(* IEC 61131-3 sources: conversion/src/times, 5 files *)

(* ---- types.st ---- *)
NAMESPACE Simatic.Ax.Conversion.Times

    TYPE
        SimotionDateTime : STRUCT
            SimotionDate : DWORD;
            SimotionTime : DWORD;
        END_STRUCT;
    END_TYPE

END_NAMESPACE

(* ---- LDateAndTimeToSimotionDateToD.st ---- *)
USING System.DateTime;
NAMESPACE Simatic.Ax.Conversion.Times
    FUNCTION LDateAndTimeToSimotionDateTime
        VAR_INPUT
            SimaticTime : LDATE_AND_TIME;
        END_VAR
        VAR_OUTPUT
            SimotionTime : DWORD;
            SimotionDate : DWORD;
        END_VAR

        VAR_TEMP
            actDays : INT;
            actMonth : INT;
            actYear : INT;
            actHour : INT;
            actMinute : INT;
            actSecond : INT;
            actMillisecond : INT;
            elapsedYears : INT;
            elapsedDays : DINT;
            loop : DINT;
        END_VAR

        //we ignore microseconds and nanoseconds, since they are supported by the destination data type
        SplitDateAndTime(value := SimaticTime,
        year => actYear,
        month => actMonth,
        day => actDays,
        hour => actHour,
        minute => actMinute,
        second => actSecond,
        millisecond => actMillisecond);

        //add number of days from full years, subtracting the current year
        FOR loop := 1992 TO (actYear - 1) DO
            IF loop MOD 4 = 0 AND loop <> 2100 THEN
                elapsedDays := elapsedDays + 366;
            ELSE
                elapsedDays := elapsedDays + 365;
            END_IF;
        END_FOR;

        //add days from full months of the current year
        IF actMonth > 1 THEN
            elapsedDays := elapsedDays + 31;
        END_IF;
        IF actMonth > 2 THEN
            IF actYear MOD 4 = 0 AND NOT (actYear = 2100) THEN
                elapsedDays := elapsedDays + 29;
            ELSE
                elapsedDays := elapsedDays + 28;
            END_IF;
        END_IF;
        IF actMonth > 3 THEN
            elapsedDays := elapsedDays + 31;
        END_IF;
        IF actMonth > 4 THEN
            elapsedDays := elapsedDays + 30;
        END_IF;
        IF actMonth > 5 THEN
            elapsedDays := elapsedDays + 31;
        END_IF;
        IF actMonth > 6 THEN
            elapsedDays := elapsedDays + 30;
        END_IF;
        IF actMonth > 7 THEN
            elapsedDays := elapsedDays + 31;
        END_IF;
        IF actMonth > 8 THEN
            elapsedDays := elapsedDays + 31;
        END_IF;
        IF actMonth > 9 THEN
            elapsedDays := elapsedDays + 30;
        END_IF;
        IF actMonth > 10 THEN
            elapsedDays := elapsedDays + 31;
        END_IF;
        IF actMonth > 11 THEN
            elapsedDays := elapsedDays + 30;
        END_IF;

        //add days from current month
        elapsedDays := elapsedDays + actDays;

        SimotionDate := TO_DWORD(elapsedDays);
        SimotionTime := TO_DWORD (TO_UDINT(actMillisecond) + UDINT#1000 * (TO_UDINT(actSecond) + UDINT#60 * (TO_UDINT(actMinute + 60 * ( actHour)))));

    END_FUNCTION

END_NAMESPACE

(* ---- SimotionDateToDToLDateAndTime.st ---- *)
USING System.DateTime;
NAMESPACE Simatic.Ax.Conversion.Times

    FUNCTION SimotionDateTimeToLDateAndTime : LDATE_AND_TIME

        VAR_INPUT
         SimotionTime : DWORD;
         SimotionDate : DWORD;
        END_VAR

        VAR_TEMP
           u32Date : UDINT;
           u32Year : UDInt;
           u32Month : UDInt;
           u32Days : UDInt;
           b32AuxHours : UDInt;
           boDateReady : Bool;
           HOUR : UDINT;
           MINUTE : UDINT;
           SECOND : UDINT;
           NANOSECOND : UDINT;
        END_VAR

        u32Date := TO_UDINT(SimotionDate);// + UDINT#1;

         // calculation of hours
         HOUR := TO_UDINT(SimotionTime) / UDINT#3600000;
         b32AuxHours := TO_UDINT(SimotionTime) - HOUR * UDINT#3600000;

         // calculation of minutes
         MINUTE := b32AuxHours / UDINT#60000;

         // calculation of seconds
         SECOND :=  (b32AuxHours - MINUTE * UDINT#60000) / UDINT#1000;

         // calculation of mseconds
         NANOSECOND := ( TO_UDINT(SimotionTime) - (HOUR *  UDINT#3600000) - (MINUTE *  UDINT#60000) - (SECOND *  UDINT#1000)) *  UDINT#1000000;

         //Reset values to calculate actual year
         u32Year :=  UDINT#1991;
         u32Days :=  UDINT#0;

         //Detect actual year by adding the days since 01.01.1992
         REPEAT
           //Increase number of years
           u32Year := u32Year +  UDINT#1;
           //If year is a leap-year
           IF  (u32Year MOD  UDINT#4 =  UDINT#0) AND  (u32Year <>  UDINT#2100) THEN //only 2100 is not a leap-year between 1992-2200
             u32Days := u32Days +  UDINT#366;
           ELSE
             u32Days := u32Days +  UDINT#365;
           END_IF;
           //Number of days is greater or equals number of days of SIMOTION system
         UNTIL u32Days >= u32Date
         END_REPEAT;

         u32Days := u32Days;

         //Decrease number of days by number of days of one year
         //If year is a leap-year
         IF  (u32Year MOD  UDINT#4 =  UDINT#0) AND  (u32Year <>  UDINT#2100) THEN //only 2100 is not a leap-year between 1992-2200
           u32Date := u32Date -  (u32Days -  UDINT#366);
         ELSE
           u32Date := u32Date -  (u32Days -  UDINT#365);
         END_IF;

         //Reset values to calculate actual month and day
         u32Month :=  UDINT#1;
         boDateReady := FALSE;

         //Start CASE with value "1" (-> january)
         REPEAT
           CASE u32Month OF
               // for months with 31 days
               UDINT#1,  UDINT#3,  UDINT#5,  UDINT#7,  UDINT#8,  UDINT#10:
               IF  (u32Date <=  UDINT#31) THEN
                 u32Days := u32Date;
                 boDateReady := TRUE;
               ELSE
                 u32Month := u32Month +  UDINT#1;
                 u32Date := u32Date -  UDINT#31;
               END_IF;
               //for february
               UDINT#2:
               IF  (u32Year MOD  UDINT#4 =  UDINT#0) AND  (u32Year <>  UDINT#2100) THEN //only 2100 is not a leap-year between 1992-2200
                 IF  (u32Date <=  UDINT#29) THEN
                   u32Days := u32Date;
                   boDateReady := TRUE;
                 ELSE
                   u32Month := u32Month +  UDINT#1;
                   u32Date := u32Date -  UDINT#29;
                 END_IF;
               ELSE
                 IF  (u32Date <=  UDINT#28) THEN
                   u32Days := u32Date;
                   boDateReady := TRUE;
                 ELSE
                   u32Month := u32Month +  UDINT#1;
                   u32Date := u32Date -  UDINT#28;
                 END_IF;
               END_IF;
               //for months with 30 days
               UDINT#4,  UDINT#6,  UDINT#9,  UDINT#11:
               IF  (u32Date <=  UDINT#30) THEN
                 u32Days := u32Date;
                 boDateReady := TRUE;
               ELSE
                 u32Month := u32Month +  UDINT#1;
                 u32Date := u32Date -  UDINT#30;
               END_IF;
               //for december
               UDINT#12:
               u32Days := u32Date;
               boDateReady := TRUE;
           END_CASE;
           //Correct month and day found
         UNTIL boDateReady = TRUE
         END_REPEAT;

         NewDateAndTime(
                     year := to_int(u32Year),
                     month := to_int(u32Month),
                     day := to_int(u32Days),
                     hour := to_int(hour),
                     minute := to_int(MINUTE),
                     second := to_int(second),
                     millisecond := to_int(NANOSECOND/UDINT#1000000),
                     value => SimotionDateTimeToLDateAndTime);

    END_FUNCTION

END_NAMESPACE

(* ---- ToLDateAndTime.st ---- *)
USING System.DateTime;

NAMESPACE Simatic.Ax.Conversion.Times

    /// Converts a SimotionDateTime structure to an LDATE_AND_TIME value.
    ///
    /// This function converts a `SimotionDateTime` structure into a Simatic `LDATE_AND_TIME` value.
    /// The date is calculated based on the number of days since 01.01.1992, and the time is derived
    /// from the number of milliseconds since midnight.
    ///
    /// @param SimotionDateTime The input SimotionDateTime structure.
    /// @return An LDATE_AND_TIME value representing the input date and time.
    {axcode:docs-v0:@simatic-ax/conversion:Times.md}
    FUNCTION ToLDateAndTime : LDATE_AND_TIME

        VAR_INPUT
         SimotionDateTime : SimotionDateTime;
        END_VAR

        VAR_TEMP
           u32Date : UDINT;
           u32Year : UDInt;
           u32Month : UDInt;
           u32Days : UDInt;
           b32AuxHours : UDInt;
           boDateReady : Bool;
           HOUR : UDINT;
           MINUTE : UDINT;
           SECOND : UDINT;
           NANOSECOND : UDINT;
        END_VAR

        u32Date := TO_UDINT(SimotionDateTime.SimotionDate);// + UDINT#1;

         // calculation of hours
         HOUR := TO_UDINT(SimotionDateTime.SimotionTime) / UDINT#3600000;
         b32AuxHours := TO_UDINT(SimotionDateTime.SimotionTime) - HOUR * UDINT#3600000;

         // calculation of minutes
         MINUTE := b32AuxHours / UDINT#60000;

         // calculation of seconds
         SECOND :=  (b32AuxHours - MINUTE * UDINT#60000) / UDINT#1000;

         // calculation of mseconds
         NANOSECOND := ( TO_UDINT(SimotionDateTime.SimotionTime) - (HOUR *  UDINT#3600000) - (MINUTE *  UDINT#60000) - (SECOND *  UDINT#1000)) *  UDINT#1000000;

         //Reset values to calculate actual year
         u32Year :=  UDINT#1991;
         u32Days :=  UDINT#0;

         //Detect actual year by adding the days since 01.01.1992
         REPEAT
           //Increase number of years
           u32Year := u32Year +  UDINT#1;
           //If year is a leap-year
           IF  (u32Year MOD  UDINT#4 =  UDINT#0) AND  (u32Year <>  UDINT#2100) THEN //only 2100 is not a leap-year between 1992-2200
             u32Days := u32Days +  UDINT#366;
           ELSE
             u32Days := u32Days +  UDINT#365;
           END_IF;
           //Number of days is greater or equals number of days of SIMOTION system
         UNTIL u32Days >= u32Date
         END_REPEAT;

         u32Days := u32Days;

         //Decrease number of days by number of days of one year
         //If year is a leap-year
         IF  (u32Year MOD  UDINT#4 =  UDINT#0) AND  (u32Year <>  UDINT#2100) THEN //only 2100 is not a leap-year between 1992-2200
           u32Date := u32Date -  (u32Days -  UDINT#366);
         ELSE
           u32Date := u32Date -  (u32Days -  UDINT#365);
         END_IF;

         //Reset values to calculate actual month and day
         u32Month :=  UDINT#1;
         boDateReady := FALSE;

         //Start CASE with value "1" (-> january)
         REPEAT
           CASE u32Month OF
               // for months with 31 days
               UDINT#1,  UDINT#3,  UDINT#5,  UDINT#7,  UDINT#8,  UDINT#10:
               IF  (u32Date <=  UDINT#31) THEN
                 u32Days := u32Date;
                 boDateReady := TRUE;
               ELSE
                 u32Month := u32Month +  UDINT#1;
                 u32Date := u32Date -  UDINT#31;
               END_IF;
               //for february
               UDINT#2:
               IF  (u32Year MOD  UDINT#4 =  UDINT#0) AND  (u32Year <>  UDINT#2100) THEN //only 2100 is not a leap-year between 1992-2200
                 IF  (u32Date <=  UDINT#29) THEN
                   u32Days := u32Date;
                   boDateReady := TRUE;
                 ELSE
                   u32Month := u32Month +  UDINT#1;
                   u32Date := u32Date -  UDINT#29;
                 END_IF;
               ELSE
                 IF  (u32Date <=  UDINT#28) THEN
                   u32Days := u32Date;
                   boDateReady := TRUE;
                 ELSE
                   u32Month := u32Month +  UDINT#1;
                   u32Date := u32Date -  UDINT#28;
                 END_IF;
               END_IF;
               //for months with 30 days
               UDINT#4,  UDINT#6,  UDINT#9,  UDINT#11:
               IF  (u32Date <=  UDINT#30) THEN
                 u32Days := u32Date;
                 boDateReady := TRUE;
               ELSE
                 u32Month := u32Month +  UDINT#1;
                 u32Date := u32Date -  UDINT#30;
               END_IF;
               //for december
               UDINT#12:
               u32Days := u32Date;
               boDateReady := TRUE;
           END_CASE;
           //Correct month and day found
         UNTIL boDateReady = TRUE
         END_REPEAT;

         NewDateAndTime(
                     year := to_int(u32Year),
                     month := to_int(u32Month),
                     day := to_int(u32Days),
                     hour := to_int(hour),
                     minute := to_int(MINUTE),
                     second := to_int(second),
                     millisecond := to_int(NANOSECOND/UDINT#1000000),
                     value => ToLDateAndTime);

    END_FUNCTION

END_NAMESPACE

(* ---- ToSimotionDateTime.st ---- *)
USING System.DateTime;

NAMESPACE Simatic.Ax.Conversion.Times

    /// Converts an LDATE_AND_TIME value to a SimotionDateTime structure.
    ///
    /// This function converts a Simatic `LDATE_AND_TIME` value into a `SimotionDateTime` structure.
    /// The date is represented as the number of days since 01.01.1992, and the time is represented
    /// as the number of milliseconds since midnight.
    ///
    /// @param SimaticTime The input LDATE_AND_TIME value.
    /// @return A SimotionDateTime structure representing the input date and time.
    {axcode:docs-v0:@simatic-ax/conversion:Times.md}
    FUNCTION ToSimotionDateTime : SimotionDateTime
        VAR_INPUT
            SimaticTime : LDATE_AND_TIME;
        END_VAR

        VAR_TEMP
            actDays : INT;
            actMonth : INT;
            actYear : INT;
            actHour : INT;
            actMinute : INT;
            actSecond : INT;
            actMillisecond : INT;
            elapsedYears : INT;
            elapsedDays : DINT;
            loop : DINT;
        END_VAR

        //we ignore microseconds and nanoseconds, since they are supported by the destination data type
        SplitDateAndTime(value := SimaticTime,
        year => actYear,
        month => actMonth,
        day => actDays,
        hour => actHour,
        minute => actMinute,
        second => actSecond,
        millisecond => actMillisecond);

        //add number of days from full years, subtracting the current year
        FOR loop := 1992 TO (actYear - 1) DO
            IF loop MOD 4 = 0 AND loop <> 2100 THEN
                elapsedDays := elapsedDays + 366;
            ELSE
                elapsedDays := elapsedDays + 365;
            END_IF;
        END_FOR;

        //add days from full months of the current year
        IF actMonth > 1 THEN
            elapsedDays := elapsedDays + 31;
        END_IF;
        IF actMonth > 2 THEN
            IF actYear MOD 4 = 0 AND NOT (actYear = 2100) THEN
                elapsedDays := elapsedDays + 29;
            ELSE
                elapsedDays := elapsedDays + 28;
            END_IF;
        END_IF;
        IF actMonth > 3 THEN
            elapsedDays := elapsedDays + 31;
        END_IF;
        IF actMonth > 4 THEN
            elapsedDays := elapsedDays + 30;
        END_IF;
        IF actMonth > 5 THEN
            elapsedDays := elapsedDays + 31;
        END_IF;
        IF actMonth > 6 THEN
            elapsedDays := elapsedDays + 30;
        END_IF;
        IF actMonth > 7 THEN
            elapsedDays := elapsedDays + 31;
        END_IF;
        IF actMonth > 8 THEN
            elapsedDays := elapsedDays + 31;
        END_IF;
        IF actMonth > 9 THEN
            elapsedDays := elapsedDays + 30;
        END_IF;
        IF actMonth > 10 THEN
            elapsedDays := elapsedDays + 31;
        END_IF;
        IF actMonth > 11 THEN
            elapsedDays := elapsedDays + 30;
        END_IF;

        //add days from current month
        elapsedDays := elapsedDays + actDays;

        ToSimotionDateTime.SimotionDate := TO_DWORD(elapsedDays);
        ToSimotionDateTime.SimotionTime := TO_DWORD (TO_UDINT(actMillisecond) + UDINT#1000 * (TO_UDINT(actSecond) + UDINT#60 * (TO_UDINT(actMinute + 60 * ( actHour)))));

    END_FUNCTION

END_NAMESPACE
